// TwinCAT 3 PLC project MyApplication
// Title: MyApplication
// Company: MyCompany
// ProjectVersion: 1.0.0.0
// ProgramVersion: 3.1.4026.18
// libraries:
//   Pushover, 1.2.0.0 (Stefan Besler)
//   Tc2_Standard, 3.4.5.0 (Beckhoff Automation GmbH)
//   Tc2_System, 3.6.4.0 (Beckhoff Automation GmbH)
//   Tc3_Module, 3.4.5.0 (Beckhoff Automation GmbH)
//   Testbench, 1.0.0.0 (Zeugwerk GmbH)
// project tree:
//   / PlcTask.TcTTO
//   POUs/ MAIN.TcPOU, Math.TcPOU
//   _Tests/ MathTest.TcPOU
// real-time tasks:
//   TASK PlcTask: cycle T#10ms, priority 20, ADS port 350
// I/O:
//   DEVICE Device 1 (EtherCAT) (disabled), AmsNetId 10.0.2.15.2.1

CONFIGURATION MyApplication
    RESOURCE PLC ON TwinCAT3
        TASK PlcTask(INTERVAL := T#10ms, PRIORITY := 20);
        PROGRAM MAIN WITH PlcTask : MAIN;
    END_RESOURCE
END_CONFIGURATION

// ---- POUs/MAIN.TcPOU
/// doc
PROGRAM MAIN
VAR
  _variant : STRING := 'Default';
  _firstCycle : BOOL := TRUE;
  _pushover : Pushover.PushoverClient('my-token', 'my-user');
  _message : STRING(255);
  _unusedButLoved : INT;
END_VAR

IF _firstCycle
THEN
  _firstCycle := FALSE;
  _message := CONCAT(CONCAT('Application using variant ', _variant), ' started');
  _pushover.SendMessageAsync('MyApplication', _message);
END_IF

_pushover.Cyclic();

END_PROGRAM

// ---- POUs/Math.TcPOU
PROGRAM Math
VAR
END_VAR

METHOD AddInt : INT
VAR_INPUT
  a : INT;
  b : INT;
END_VAR
AddInt := a + b;
END_METHOD

END_PROGRAM

// ---- _Tests/MathTest.TcPOU
FUNCTION_BLOCK MathTest IMPLEMENTS Testbench.IUnitTest;

METHOD Test_GivenTwoIntegers_WhenAddInt_SumIsCalculated
VAR_INPUT
  assertions : Testbench.IAssertions;
END_VAR
VAR
  result : INT;
END_VAR
result := Math.AddInt(5, 6);

assertions.EqualsInt(expected := 11, actual := result, '5+6=11');
END_METHOD

END_FUNCTION_BLOCK
